% RSLogix 500 project 9.1.RSS, saved by version 8.30.00.16 %
PROJECT "9.1"    % processor: Bul.1763 MicroLogix 1100 Series B %

PROGRAM FILES
  LAD 2   10 rungs

DATA FILES
  O0 OUTPUT  4 elements
  I1 INPUT  6 elements
  S2 STATUS  66 elements
  B3 BINARY  2 elements
  T4 TIMER  1 elements
  C5 COUNTER  1 elements
  R6 CONTROL  1 elements
  N7 INTEGER  4 elements
  F8 FLOAT  1 elements

LADDER 2
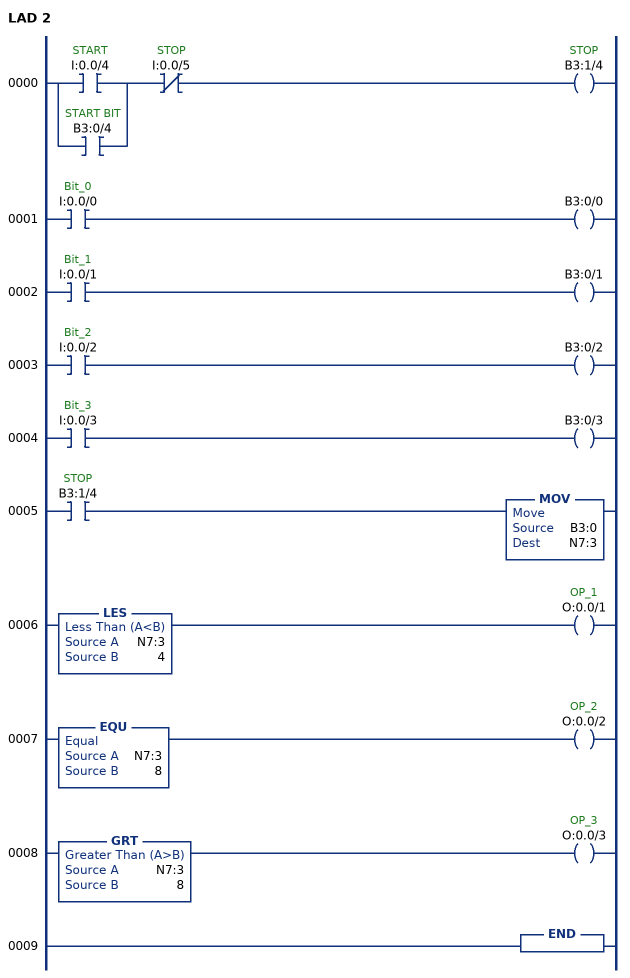
% Rung: 0 %
SOR BST XIC I:0.0/4 NXB XIC B3:0/4 BND XIO I:0.0/5 OTE B3:1/4 EOR
%   I:0.0/4  "START" %
%   B3:0/4  "START BIT" %
%   I:0.0/5  "STOP" %
%   B3:1/4  "STOP" %
% Rung: 1 %
SOR XIC I:0.0/0 OTE B3:0/0 EOR
%   I:0.0/0  "Bit_0" %
% Rung: 2 %
SOR XIC I:0.0/1 OTE B3:0/1 EOR
%   I:0.0/1  "Bit_1" %
% Rung: 3 %
SOR XIC I:0.0/2 OTE B3:0/2 EOR
%   I:0.0/2  "Bit_2" %
% Rung: 4 %
SOR XIC I:0.0/3 OTE B3:0/3 EOR
%   I:0.0/3  "Bit_3" %
% Rung: 5 %
SOR XIC B3:1/4 MOV B3:0 N7:3 EOR
%   B3:1/4  "STOP" %
% Rung: 6 %
SOR LES N7:3 4 OTE O:0.0/1 EOR
%   O:0.0/1  "OP_1" %
% Rung: 7 %
SOR EQU N7:3 8 OTE O:0.0/2 EOR
%   O:0.0/2  "OP_2" %
% Rung: 8 %
SOR GRT N7:3 8 OTE O:0.0/3 EOR
%   O:0.0/3  "OP_3" %
% Rung: 9 %
SOR END EOR
